Fanuc KAREL source: DEF_SCREEN.kl

PROGRAM T
%NOLOCKGROUP
VAR
 v0 : STRING[40]
 v1 : STRING[40]
 v2 : INTEGER
BEGIN
 DEF_SCREEN(v0, v1, v2)
END T
